Fanuc KAREL source: kt00501.KL

PROGRAM KT00501
%STACKSIZE=65535
%PRIORITY=65535
%NOLOCKGROUP
VAR
P1 : XYZWPR
P2 : XYZWPR
OUT : XYZWPREXT
BEGIN
P1.X=1.0
P2.Y=2.0
P1.X=1.0
P2.Y=2.0
-- UNRESOLVED_PC line 12 opcodes [49 7E 49 7E 60 7E 4A] marker_code=80
END KT00501
